FUNCTION FC_OeeSetUpdateCount
VAR_INPUT
	aByte					: stByteAsBit;
END_VAR

IF FC_ProductStatusNopresence(aByte) = eProductStatus.Completed THEN
	G.OEE_bCountUpGood := TRUE;
END_IF
IF FC_ProductStatusNopresence(aByte) = eProductStatus.Scraped THEN
	G.OEE_bCountUpBad := TRUE;
END_IF

END_FUNCTION

(* stored: Version 1.1.0.1, ProductVersion 3.1.4024.15
   POU FC_OeeSetUpdateCount: Id {1f06fba6-34a1-46a6-ad32-2f2eab99a685}, SpecialFunc None *)
